// TIA Portal V20 export
// export: Created 2025-12-01T14:57:11.8627361Z, ExportSetting None, DisplayName Totally Integrated Automation Portal, DisplayVersion V20 Update 3, DisplayName TIA Portal Openness, DisplayVersion V20 Update 3, DisplayName TIA Portal Version Control Interface, DisplayVersion V20 Update 3, DisplayName STEP 7 Professional, DisplayVersion V20 Update 3, DisplayName STEP 7 Safety, DisplayVersion V20 Update 2, DisplayName WinCC Basic/Comfort/Advanced, DisplayVersion V20 Update 3, DisplayName WinCC Professional, DisplayVersion V20 Update 3, DisplayName WinCC Unified, DisplayVersion V20 Update 3
FUNCTION "FC770_Control_ApiladorCajasPlastico" : Void   // FC770, STL
TITLE = Orden a generar para el Apilador de Cajas
{ S7_Optimized_Access := 'FALSE' }
AUTHOR : TRACKING
NAME : 20141014
VERSION : 4.0
// stored: AutoNumber false
   VAR_INPUT
      EstadoZonaMaquina : "EstadoZona";   // Status de la Maquina (ZONA)
      EstadoZonaMesa : "EstadoZona";   // Status de la Mesa (ZONA)
      MesaVI : UInt;   // Mesa Asociada a la Maquina
      MesaVI_Anterior : UInt;   // Mesa Anterior
      Offset : UInt;   // Offset desde Poscion 0 hasta la Posicion Banda (+ / -)
      OrdenUT_MAnt : Bool;   // Orden de Salida de la UT de la Mesa Anterior
      AcabadaOrden : Bool;   // Orden Acabada de la Maquina
   END_VAR
   VAR_IN_OUT
      PosInicial : UInt;   // Dato 01 de la Maquina : Posición de Recogida
      PosFinal : UInt;   // Dato 02 de la Maquina : Posición de Acabada
      TipoAmarre : UInt;   // Dato 03 de la Maquina : Tipo de Amarre
      PosPreviaInicial : UInt;   // Dato 04 de la Maquina: Posicion Previa de Recogida
      RealizarOrden : Bool;   // Realizar la orden de la Maquina
   END_VAR
   VAR_TEMP
      NumeroUT_01 : UInt;
      NumeroUT_02 : UInt;
      NumeroUT : UInt;
      SiguienteUT : UInt;
      AlturaF01 : UInt;
      AmarreF01 : UInt;
      AlturaF02 : UInt;
      AmarreF02 : UInt;
      CuantasUT : UInt;
   END_VAR
BEGIN

NETWORK
TITLE = Inicializaciones
/////////////////////////////////////////////////////////////////////////////
// ---  Inicializar Variables

      L     0;
      T     #AlturaF01;
      T     #AlturaF02;
      T     #AmarreF02;
      T     #CuantasUT;

      L     90;
      T     #AmarreF01;  // Por si esta vacio



NETWORK
TITLE = Reset de Variables
/////////////////////////////////////////////////////////////////////////////
// --- Si realiza un reset hay que limpiar las variables

      AN    #EstadoZonaMaquina.PerReset_CBx;
      JC    NoExiste_Reset;  // Reseteada la Maquina

      SET;
      R     #RealizarOrden;  // Resetear la orden enviada

      L     0;
      T     #PosInicial;
      T     #PosFinal;
      T     #TipoAmarre;
      T     #PosPreviaInicial;

      JU    Final;  // Finalizado el tratamiento de la Maquina

NoExiste_Reset:NOP   0;



NETWORK
TITLE = Distribución
// - Inicialiar Variables
// - Cierre del protocolo de la orden
// - Calcular la orden
/////////////////////////////////////////////////////////////////////////////
// --- Mirar si necesita calcular orden  y cerrar protocolos

      A     #OrdenUT_MAnt;
      AN    #RealizarOrden;
      AN    #AcabadaOrden;
      JC    CalcularOperacion_DelApilador;  // Nueva Orden a Realizar ?

      A     #AcabadaOrden;
      A     #RealizarOrden;  // Ya hay que finalizar la Orden ?
      JCN   Final;

      SET;
      R     #RealizarOrden;  // Resetear la orden enviada

      L     0;
      T     #PosInicial;
      T     #PosFinal;
      T     #TipoAmarre;
      T     #PosPreviaInicial;

      JU    Final;  // Finalizado el tratamiento de la Maquina



NETWORK
TITLE = Calcular la Orden para la Maquina
CalcularOperacion_DelApilador:NOP   0;

/////////////////////////////////////////////////////////////////////////////
// --- Comprobación primera --> PosInicial, PosFinal, TipoAmarre

      L     #PosInicial;
      L     0;
      <>I;
      JC    Final;

      L     #PosFinal;
      L     0;
      <>I;
      JC    Final;

      L     #TipoAmarre;
      L     0;
      <>I;
      JC    Final;

      L     #PosPreviaInicial;
      L     0;
      <>I;
      JC    Final;

/////////////////////////////////////////////////////////////////////////////
// --- En Marcha y sin error ==> Maquina y Mesa

      A     #EstadoZonaMaquina.Marcha_CBx;
      AN    #EstadoZonaMaquina.Error_CBx;
      A     #EstadoZonaMesa.Marcha_CBx;
      AN    #EstadoZonaMesa.Error_CBx;
      JCN   Final;


/////////////////////////////////////////////////////////////////////////////
/////////////////////////////////////////////////////////////////////////////
// ---
// ---                  CALCULO DE LA ORDEN
// ---
/////////////////////////////////////////////////////////////////////////////
/////////////////////////////////////////////////////////////////////////////



NETWORK
TITLE = Datos de las UT's de Mesa de Maquina
/////////////////////////////////////////////////////////////////////////////
// ---  Recoger los Datos de la Mesa de la Maquina

      L     "DB810_ColasMesas".Colas[#MesaVI].UT_PrimeraMesa;
      T     #SiguienteUT;

      L     #SiguienteUT;
      L     0;
      ==I;
      JC    RecogerDatos_MesaAnterior;  // No hay UT's, Esta Vacia ?


/////////////////////////////////////////////////////////////////////////////I
// --- Buscar la Ultima UT

BucleBusquedaUltimaUT_DeMesa:NOP   0;
      L     #SiguienteUT;
      T     #NumeroUT;

      L     "DB812_UTs_Control".UT[#NumeroUT].UT_SiguienteMesa;
      T     #SiguienteUT;

      L     #SiguienteUT;
      L     0;
      <>I;
      JC    BucleBusquedaUltimaUT_DeMesa;  // Es la Ultima UT ?

      L     #NumeroUT;
      T     #NumeroUT_01;
      L     "DB815_UTs_Datos".UT[#NumeroUT_01].CotaAltura;
      T     #AlturaF01;
      L     "DB815_UTs_Datos".UT[#NumeroUT_01].Amarre;
      T     #AmarreF01;


/////////////////////////////////////////////////////////////////////////////
// --- Identico Amarre entre Pequenas y Grandes
// --- Identico Amarre entre Pequenas y Grandes (Diferente en EUROPOOL)
// --- No hay que calcular cuantas hay en la Fila

//      SPA   RecogerDatos_MesaAnterior


/////////////////////////////////////////////////////////////////////////////
// --- Cambio de funcionamiento en Tipo de Amarre que se envia
// --- Caja Grande --> TipoAmarre = 0
// --- Caja Pequeña --> TipoAmarre = 1 ( Da lo mismo Doble que Simple)

      L     0;
      T     #CuantasUT;  // Caja Grande --> TipoAmarre = 0

      L     "DB812_UTs_Control".UT[#NumeroUT].TipoCarga;
      L     10;
      /I;
      L     11;  // CA_2 (Caja Grande)
      ==I;
      JC    RecogerDatos_MesaAnterior;

      L     1;
      T     #CuantasUT;  // Caja Pequeña --> TipoAmarre = 1
      JU    RecogerDatos_MesaAnterior;



NETWORK
TITLE = Datos de las UT's de Mesa Anterior a la Maquina
RecogerDatos_MesaAnterior:NOP   0;

/////////////////////////////////////////////////////////////////////////////
// --- Recoger los Datos de la Mesa Anterior a la Maquina

      L     "DB810_ColasMesas".Colas[#MesaVI_Anterior].UT_PrimeraMesa;
      T     #NumeroUT_02;

      L     "DB815_UTs_Datos".UT[#NumeroUT_02].CotaAltura;
      T     #AlturaF02;
      L     "DB815_UTs_Datos".UT[#NumeroUT_02].Amarre;
      T     #AmarreF02;



NETWORK
TITLE = Calculo Final de Orden para la Maquina
/////////////////////////////////////////////////////////////////////////////
/////////////////////////////////////////////////////////////////////////////
// --- Realizar el Calculo Final
// ---      Posicion Inicial
// ---      Posicion Final
// ---      Tipo de Arrarre


/////////////////////////////////////////////////////////////////////////////
// --- Posicion Inicial = AmarreF01
      L     #AmarreF01;  // PosInicial = AmarreF01
      L     #Offset;  // + Offset de Desapilador
      +I;
      T     #PosInicial;

/////////////////////////////////////////////////////////////////////////////
// --- Posicion Final = AmarreF01 + AlturaF02 - 3

      L     #AlturaF02;  // PosFinal = (AmarreF01 + AlturaF02 - 3)
      L     #AmarreF01;
      +I;
      L     3;
      -I;
      L     #Offset;  // + Offset de Desapilador
      +I;
      T     #PosFinal;

/////////////////////////////////////////////////////////////////////////////
// --- Posicion Previa Inicial = AmarreF02

      L     #AmarreF02;
      L     #Offset;  // + Offset de Desapilador
      +I;
      T     #PosPreviaInicial;

/////////////////////////////////////////////////////////////////////////////
// --- Calculo de la TipoAmarre

      L     #CuantasUT;
      T     #TipoAmarre;

/////////////////////////////////////////////////////////////////////////////
// --- Activar Orden

      SET;
      S     #RealizarOrden;  // Activacion de la Orden



NETWORK
TITLE = Finalizar la función
/////////////////////////////////////////////////////////////////////////////
// --- Finalizado el tratamiento de la Orden
Final:NOP   0;


END_FUNCTION
